INTERFACE ITaskContainer

PROPERTY Lock : INT
GET
END_GET
SET
END_SET
END_PROPERTY

END_INTERFACE

(* stored: Version 1.1.0.1, ProductVersion 3.1.4024.5
   Itf ITaskContainer: Id {f8f0b8c8-1cba-4926-b45f-a93038fb862d}
   Property Lock: Id {b1f770b0-0ea3-49e1-b348-e1d7cbaaf8c2}
   Get Get: Id {16a834ee-b5ac-4a70-8236-cfe370817a40}
   Set Set: Id {52d25b29-5880-42cf-bbea-f5fb93f2dba2} *)
